(* PLC project Generated.project, CODESYS CODESYS V3.5 SP19 Patch 1 *)
(* stored: creationDateTime 2026-09-01T01:00:08.898708, modificationDateTime 2026-09-01T01:00:08.898708 *)

(* ═══════════════════════════════════════════════════════════════ ⚙️ ST_CycleExtractionCfg — Réglages persistants cycle extraction 📄 Doc : DOC/AF/AF_Partie-04_Mode_SemiAuto_Sequenceur_v2.3.md §3ter ═══════════════════════════════════════════════════════════════ *)
TYPE ST_CycleExtractionCfg : STRUCT
  ExtractionControlDistance_M : REAL := 2;  (* Remontée palier 1 avant accélération *)
  Initialized : BOOL := FALSE;  (* 🚦 flag restauration boot *)
END_STRUCT;
END_TYPE
